// TIA Portal V19 export
TYPE "UDT_STATUS_TANK"
   STRUCT
      isAllowedToFill : Bool;
      isAllowedToEmpty : Bool;
      isFilling : Bool;
      isGettingEmpty : Bool;
   END_STRUCT;
END_TYPE
